(* IEC 61131-3 sources: CodesysTest/alpha/export/Device.dev/Plc Logic/Application/ObjectHandling/FB_CollectionHandlerExecutable.pou, 1 file *)

(* ---- FB_CollectionHandlerExecutable.pou.st ---- *)
(*#-#-#-#-#-#-#-#-#-#---Declaration---#-#-#-#-#-#-#-#-#-#-#-#-#*)

FUNCTION_BLOCK FB_CollectionHandlerExecutable
VAR_INPUT
END_VAR
VAR
	Collection: ARRAY[0..GlobalObjects.MAX_EXECUTEABLE] OF IExecuteAutomatically; // object array
	ObjNames   : ARRAY[0..GlobalObjects.MAX_EXECUTEABLE] OF STRING;
	_ArrayOver   : BOOL;
	_BadObj      : INT;
	_DupeObj   : INT;
	_OverObj   : INT;
	_TotalObj   : UINT;
END_VAR(*#-#-#-#-#-#-#-#-#-#---Implementation---#-#-#-#-#-#-#-#-#-#-#-#-#*)

//	Function Block: FB_CollectionHandlerExecutable
//	Description: This collection handler stores executable FB's to an array
//				 and has a method to execute them all on demand
//	Created by: Ben Hess
//	Created Date: Friday, September 7, 2018
